# B&R Automation Studio project Panasonic_LinkaPowerCP2_A2021055 (part 16)

#### Main.st - Init, cyclic, exit code
```iecst
PROGRAM _INIT
	(* Insert code here *)

END_PROGRAM

PROGRAM _CYCLIC

	//Volanie funkcie SequenceControl//
	SequenceControl(SC:= SC_P2_StoperZaklTesnenia);

	//Volanie podprogramov//
	IOLinkKomunikacia;

	//Zhasnutie Bannera//
	IF P2_StoperZaklTesnenia.CMD.Banner_LED_OFF THEN
		P2_StoperZaklTesnenia.Banner.IN.ModraLED_ON:= FALSE;
		P2_StoperZaklTesnenia.Banner.IN.CervenaLED_ON:= FALSE;
		P2_StoperZaklTesnenia.Banner.IN.CyanLED_ON:= FALSE;
		P2_StoperZaklTesnenia.Banner.IN.ModraRotujucaLED_ON:= FALSE;
		P2_StoperZaklTesnenia.Banner.IN.OranzovaLED_ON:= FALSE;
		P2_StoperZaklTesnenia.Banner.IN.ZelenaLED_ON:= FALSE;
		P2_StoperZaklTesnenia.Banner.IN.ZltaLED_ON:= FALSE;
		P2_StoperZaklTesnenia.CMD.Banner_LED_OFF:= FALSE;
	END_IF

	//Reset sekcie //
	IF P2_StoperZaklTesnenia.Reset THEN
		SC_P2_StoperZaklTesnenia.Step:= 0;
		P2_StoperZaklTesnenia.Reset:= FALSE;
	ELSIF NOT Safety.STAV.Linka_ZonaCS_AKTIVNA THEN
		SC_P2_StoperZaklTesnenia.Step:= 0;
	END_IF

	CASE SC_P2_StoperZaklTesnenia.Step OF

		0:
			SC_P2_StoperZaklTesnenia.StepName:='0 - Nulovanie';
			P2_StoperZaklTesnenia.Automat:= FALSE;
			P2_StoperZaklTesnenia.KoniecCyklu:= FALSE;
			P2_StoperZaklTesnenia.Manual:= FALSE;
			P2_StoperZaklTesnenia.STAV.PoINIT:= FALSE;
			P2_StoperZaklTesnenia.OUT.ZasunStoper:= FALSE;
			P2_StoperZaklTesnenia.RFID_hlava.PrecitajChipRFID:= FALSE;
			P2_StoperZaklTesnenia.CMD.Banner_LED_OFF:= TRUE;
			P2_ZakladacTesnenia.COM_IN.ZalozTesnenie:= FALSE;
			P2_ZakladacTesnenia.COM_OUT.Stav_ZalozenieTesneniaUkoncene:= FALSE;
			CAM1.CMD.Triger:= FALSE;
			CAM1.STAV.Results_READY:= FALSE;
			FTP_CAM1.CMD.OdosliFotku:= FALSE;
			FTP_CAM1.CMD.VymazFotku:= FALSE;
			CAM7.CMD.Triger:= FALSE;
			CAM7.STAV.Results_READY:= FALSE;

			CAM8.CMD.Triger:= FALSE;
			CAM8.STAV.Results_READY:= FALSE;

			CAM17.CMD.Triger:= FALSE;
			CAM17.STAV.Results_READY:= FALSE;
			FTP_CAM17.CMD.OdosliFotku:= FALSE;
			FTP_CAM17.CMD.VymazFotku:= FALSE;
			P2_ZaklTesn_KAM_Result_Ignoruj:= FALSE;
			TRCB_P2_ZakladacTesnenia_ST3.CMD.VyziadajStavPaletky_TYP1:= FALSE;
			TRCB_P2_ZakladacTesnenia_ST3.CMD.PriradQRkodFiltra_TYP3:= FALSE;
			TRCB_P2_ZakladacTesnenia_ST3.CMD.OdosliStavPaletky_TYP2:= FALSE;
			TRCB_P2_ZakladacTesnenia_ST3.CMD.VyziadajStavPanatrace_TYP4:= FALSE;
			P2_Vizu.ZobrazHL1_ST3:= FALSE;
			P2_Vizu.ZobrazHL2_ST3:= FALSE;
			P2_Vizu.ZobrazHL3_ST3:= FALSE;
			P2_Vizu.ZobrazHL4_ST3:= FALSE;
			P2_Vizu.ZobrazHL5_ST3:= FALSE;
			P2_Vizu.ZobrazHL6_ST3:= FALSE;
			P2_Vizu.ZobrazHL7_ST3:= FALSE;
			P2_Vizu.ZobrazHL8_ST3:= FALSE;
			P2_Vizu.ZobrazHL9_ST3:= FALSE;
			P2_Vizu.ZobrazHL10_ST3:= FALSE;
			P2_Vizu.ZobrazHL11_ST3:= FALSE;
			P2_Vizu.ZobrazHL12_ST3:= FALSE;
			P2_Vizu.ZobrazHL14_ST3:= FALSE;
			P2_Vizu.ZobrazHL15_ST3:= FALSE;
			PocetDopytovNaServer:= 0;
			CisloFotky:= 0;
			PocetTrigrovKamery:= 0;
			P1_AkumulacnyStoper.STAV.PrebiehaVyvezeniePaletky:= FALSE;
			P2_StoperZaklTesnenia.STAV.PrebiehaVyvezeniePaletky:= FALSE;
			OpatovnaKontrolaFiltra_5H:= FALSE;
			PrecitanyQRkodPowerCP:= '';
			PrecitanyQRkodFiltra5H:= '';
			PrecitaneCisloPaletky:= '';
			TestovaciKus:= FALSE;
			P2_StoperZaklTesnenia.STAV.ObsluhaOznacilaPaletku_NG:= FALSE;
			P2_ZakladanieTesnenia_Taktime.IN.START_MeraniaCasu:= FALSE;
			P2_ZakladanieTesnenia_Taktime.IN.START_MeraniaStratovehoCasu:= FALSE;

			IF Safety.STAV.Linka_ZonaCS_AKTIVNA AND
				P2_Pracovisko.STAV.HardwareZaklTesnenia_OK AND
				NOT P2_Pracovisko.STAV.Porucha_ST1 THEN
				SC_P2_StoperZaklTesnenia.ResetStep:= TRUE;
				SC_P2_StoperZaklTesnenia.Step:= 1;
			END_IF

		1:
			SC_P2_StoperZaklTesnenia.StepName:='1 - Cakam na spustenie vyroby';
			P2_StoperZaklTesnenia.KoniecCyklu:= FALSE;
			IF P2_StoperZaklTesnenia.Automat THEN
				SC_P2_StoperZaklTesnenia.Step:= 2;
			ELSIF P2_StoperZaklTesnenia.Manual THEN
				SC_P2_StoperZaklTesnenia.Step:= 700;
			END_IF

			//********************************************************Inicializácia****************************************************************************//

		2:
			SC_P2_StoperZaklTesnenia.StepName:='2 - Inicializacia - cakam na spustenie inicializacie';
			SC_P2_StoperZaklTesnenia.IdleTime.PT:= T#4s;
			SC_P2_StoperZaklTesnenia.AlarmTime.PT:= T#5s;

			IF P2_ZakladacTesnenia.STAV.PoINIT AND P2_ZakladacTesnenia.ServoPojazduZakladaca.Status.ActPosition < 5  AND (*Safety.STAV.P2_ZaklTesn_PojazdMuting_AKTIVNY AND*) P2_Dopravniky.STAV.PoINIT THEN
				SC_P2_StoperZaklTesnenia.ResetStep:= TRUE;
				SC_P2_StoperZaklTesnenia.Step:= 3;
			END_IF

		3:
			SC_P2_StoperZaklTesnenia.StepName:='3 - Inicializacia - vymazanie adresarov kamier CAM1 a CAM 17';
			SC_P2_StoperZaklTesnenia.IdleTime.PT:= T#4s;
			SC_P2_StoperZaklTesnenia.AlarmTime.PT:= T#5s;

			P2_StoperZaklTesnenia.Banner.IN.ModraRotujucaLED_ON:= TRUE;

			IF NOT SC_P2_StoperZaklTesnenia.Switch1 THEN
				FTP_CAM1.CMD.VymazFotku:= TRUE;
				FTP_CAM17.CMD.VymazFotku:= TRUE;
				SC_P2_StoperZaklTesnenia.Switch1:= TRUE;
			END_IF

			IF FTP_CAM1.STATUS.KomunikaciaUkoncena AND FTP_CAM17.STATUS.KomunikaciaUkoncena THEN
				P2_StoperZaklTesnenia.CMD.Banner_LED_OFF:= TRUE;
				FTP_CAM1.CMD.VymazFotku:= FALSE;
				FTP_CAM17.CMD.VymazFotku:= FALSE;
				SC_P2_StoperZaklTesnenia.ResetStep:= TRUE;
				SC_P2_StoperZaklTesnenia.Step:= 5;
			ELSIF FTP_CAM1.STATUS.KomunikaciaError THEN
				P2_Alarmy[225]:= TRUE;
				P2_Pracovisko.STAV.Porucha_ST1:= TRUE;
			ELSIF FTP_CAM17.STATUS.KomunikaciaError THEN
				P2_Alarmy[228]:= TRUE;
				P2_Pracovisko.STAV.Porucha_ST1:= TRUE;
			END_IF

		5:
			SC_P2_StoperZaklTesnenia.StepName:='5 - Inicializacia - hladanie paletky na stopri';
			SC_P2_StoperZaklTesnenia.IdleTime.PT:= T#5s;
			SC_P2_StoperZaklTesnenia.AlarmTime.PT:= T#5s;

			SC_P2_StoperZaklTesnenia.IdleTime.IN:= TRUE;

			IF P2_StoperZaklTesnenia.RFID_hlava.PritomnostPaletky THEN
				SC_P2_StoperZaklTesnenia.ResetStep:= TRUE;
				SC_P2_StoperZaklTesnenia.Step:= 20;
			ELSIF SC_P2_StoperZaklTesnenia.IdleTime.Q THEN
				P2_StoperZaklTesnenia.STAV.PoINIT:= TRUE;
				SC_P2_StoperZaklTesnenia.ResetStep:= TRUE;
				SC_P2_StoperZaklTesnenia.Step:= 100;
			END_IF

		20:
			SC_P2_StoperZaklTesnenia.StepName:='20 - Inicializacia - precitanie cisla paletky';
			SC_P2_StoperZaklTesnenia.IdleTime.PT:= T#200ms;
			SC_P2_StoperZaklTesnenia.AlarmTime.PT:= T#5s;

			SC_P2_StoperZaklTesnenia.IdleTime.IN:= P2_StoperZaklTesnenia.RFID_hlava.PritomnostPaletky;

			IF SC_P2_StoperZaklTesnenia.IdleTime.Q AND NOT SC_P2_StoperZaklTesnenia.Switch1 THEN
				P2_StoperZaklTesnenia.RFID_hlava.PrecitajChipRFID:= TRUE;
				i:= 0;
				SC_P2_StoperZaklTesnenia.Switch1:= TRUE;
			END_IF

			IF P2_StoperZaklTesnenia.RFID_hlava.Stav_CitanieZapis_OK AND P2_StoperZaklTesnenia.RFID_hlava.PrecitaneCisloPaletky <> 0 THEN
				i:= P2_StoperZaklTesnenia.RFID_hlava.PrecitaneCisloPaletky;
				P2_StoperZaklTesnenia.PAR.CisloPaletky:= P2_StoperZaklTesnenia.RFID_hlava.PrecitaneCisloPaletky;
				P2_StoperZaklTesnenia.RFID_hlava.PrecitajChipRFID:= FALSE;
				SC_P2_StoperZaklTesnenia.ResetStep:= TRUE;
				SC_P2_StoperZaklTesnenia.Step:= 23;
			END_IF

		23:
			SC_P2_StoperZaklTesnenia.StepName:='23 - Inicializacia - kontrola a priradenie indexu paletky na zaklade precitanej hodnoty';
			SC_P2_StoperZaklTesnenia.IdleTime.PT:= T#200ms;
			SC_P2_StoperZaklTesnenia.AlarmTime.PT:= T#5s;

			IF i<> 0 THEN
				P2_StoperZaklTesnenia.PAR.CisloPaletky_STRING:= USINT_TO_STRING(i);
				Paletka[i].PAR.CisloPaletky:= USINT_TO_STRING(i);
				P2_ZakladacTesnenia.PAR.IndexPaletky:= i;
				SC_P2_StoperZaklTesnenia.ResetStep:= TRUE;
				SC_P2_StoperZaklTesnenia.Step:= 30;
			ELSE
				P2_Alarmy[200]:= TRUE;
				P2_Pracovisko.STAV.Porucha_ST1:= TRUE;
			END_IF

		30:
			SC_P2_StoperZaklTesnenia.StepName:='30 - Inicializacia - kontrola stavu paletky';
			SC_P2_StoperZaklTesnenia.IdleTime.PT:= T#200ms;
			SC_P2_StoperZaklTesnenia.AlarmTime.PT:= T#5s;

			IF Paletka[i].STAV.StavPaletky = '' THEN
				Paletka[i].STAV.StavPaletky:= 'NG';
				SC_P2_StoperZaklTesnenia.ResetStep:= TRUE;
				SC_P2_StoperZaklTesnenia.Step:= 560;
			ELSIF Paletka[i].STAV.StavPaletky = 'PRECH' THEN
				P2_StoperZaklTesnenia.STAV.PoINIT:= TRUE;
				SC_P2_StoperZaklTesnenia.ResetStep:= TRUE;
				SC_P2_StoperZaklTesnenia.Step:= 560;
			ELSIF Paletka[i].STAV.StavPaletky = 'TEST' AND Paletka[i].STAV.CisloTestovacejStanice = 'ST_3' THEN
				TestovaciKus:= TRUE;
			ELSIF Paletka[i].STAV.StavPaletky = 'TEST' AND Paletka[i].STAV.CisloTestovacejStanice <> 'ST_3' THEN
				P2_StoperZaklTesnenia.STAV.PoINIT:= TRUE;
				SC_P2_StoperZaklTesnenia.ResetStep:= TRUE;
				SC_P2_StoperZaklTesnenia.Step:= 560;
			ELSIF Paletka[i].STAV.StavPaletky = 'REV' AND Paletka[i].STAV.CisloRevorkovejStanice = 'ST_3' THEN
				Paletka[i].STAV.StavPaletky:= 'OK';
				SC_P2_StoperZaklTesnenia.ResetStep:= TRUE;
				SC_P2_StoperZaklTesnenia.Step:= 33;
			ELSIF Paletka[i].STAV.StavPaletky = 'REV' AND Paletka[i].STAV.CisloRevorkovejStanice <> 'ST_3' THEN
				P2_StoperZaklTesnenia.STAV.PoINIT:= TRUE;
				SC_P2_StoperZaklTesnenia.ResetStep:= TRUE;
				SC_P2_StoperZaklTesnenia.Step:= 560;
			ELSIF Paletka[i].STAV.StavPaletky = 'OK' THEN
				SC_P2_StoperZaklTesnenia.ResetStep:= TRUE;
				SC_P2_StoperZaklTesnenia.Step:= 33;
			ELSIF Paletka[i].STAV.StavPaletky = 'NG' THEN
				P2_StoperZaklTesnenia.STAV.PoINIT:= TRUE;
				SC_P2_StoperZaklTesnenia.ResetStep:= TRUE;
				SC_P2_StoperZaklTesnenia.Step:= 560;
			END_IF

		33:
			SC_P2_StoperZaklTesnenia.StepName:='33 - Inicializacia - kontrola uzavretia komunikacie';
			SC_P2_StoperZaklTesnenia.IdleTime.PT:= T#200ms;
			SC_P2_StoperZaklTesnenia.AlarmTime.PT:= T#5s;

			IF Paletka[i].STAV.Komunikacia_DONE THEN
				P2_StoperZaklTesnenia.STAV.PoINIT:= TRUE;
				SC_P2_StoperZaklTesnenia.ResetStep:= TRUE;
				SC_P2_StoperZaklTesnenia.Step:= 560;
			ELSE
				P2_StoperZaklTesnenia.STAV.PoINIT:= TRUE;
				SC_P2_StoperZaklTesnenia.ResetStep:= TRUE;
				SC_P2_StoperZaklTesnenia.Step:= 100;
			END_IF

			//********************************************************Automatický režim****************************************************************************//

		100:
			SC_P2_StoperZaklTesnenia.StepName:='100 - Automaticky Rezim - cakam na príchod paletky na stoper';
			SC_P2_StoperZaklTesnenia.IdleTime.PT:= T#200ms;
			SC_P2_StoperZaklTesnenia.AlarmTime.PT:= T#5s;

			SC_P2_StoperZaklTesnenia.IdleTime.IN:= P2_StoperZaklTesnenia.RFID_hlava.PritomnostPaletky;

			IF P2_StoperZaklTesnenia.RFID_hlava.PritomnostPaletky THEN
				P1_AkumulacnyStoper.STAV.PrebiehaVyvezeniePaletky:= FALSE;
			END_IF

			IF NOT SC_P2_StoperZaklTesnenia.Switch1 AND P2_StoperZaklTesnenia.RFID_hlava.PritomnostPaletky THEN
				P2_ZakladanieTesnenia_Taktime.IN.START_MeraniaCasu:= TRUE;
				P2_ZakladanieTesnenia_Taktime.IN.ZAPIS_MeraniaCasu:= TRUE;
				P2_ZakladanieTesnenia_Taktime.IN.ZAPIS_StratovyCas:= TRUE;
				Buffer_3.Hodnota:= P2_ZakladanieTesnenia_Taktime.OUT.StratoveSekundy;
				Buffer_3.ZapisHodnotu:= TRUE;
				SC_P2_StoperZaklTesnenia.Switch1:= TRUE;
			END_IF

			IF P2_StoperZaklTesnenia.KoniecCyklu THEN
				SC_P2_StoperZaklTesnenia.ResetStep:= TRUE;
				SC_P2_StoperZaklTesnenia.Step:= 0;
			ELSIF SC_P2_StoperZaklTesnenia.IdleTime.Q THEN
				SC_P2_StoperZaklTesnenia.ResetStep:= TRUE;
				SC_P2_StoperZaklTesnenia.Step:= 101;
			END_IF

		101:
			SC_P2_StoperZaklTesnenia.StepName:='101 - Automaticky Rezim - precitanie cisla paletky';
			SC_P2_StoperZaklTesnenia.IdleTime.PT:= T#500ms;
			SC_P2_StoperZaklTesnenia.AlarmTime.PT:= T#5s;
			SC_P2_StoperZaklTesnenia.IdleTime.IN:= TRUE;

			IF NOT SC_P2_StoperZaklTesnenia.Switch1 THEN
				i:= 0;
				P2_StoperZaklTesnenia.RFID_hlava.PrecitajChipRFID:= TRUE;
				SC_P2_StoperZaklTesnenia.Switch1:= TRUE;
			END_IF

			IF P2_StoperZaklTesnenia.RFID_hlava.Stav_CitanieZapis_OK AND P2_StoperZaklTesnenia.RFID_hlava.PrecitaneCisloPaletky <> 0 THEN
				i:= P2_StoperZaklTesnenia.RFID_hlava.PrecitaneCisloPaletky;
				P2_StoperZaklTesnenia.PAR.CisloPaletky:= P2_StoperZaklTesnenia.RFID_hlava.PrecitaneCisloPaletky;
				P2_StoperZaklTesnenia.RFID_hlava.PrecitajChipRFID:= FALSE;
				SC_P2_StoperZaklTesnenia.ResetStep:= TRUE;
				SC_P2_StoperZaklTesnenia.Step:= 102;
			END_IF

		102:
			SC_P2_StoperZaklTesnenia.StepName:='102 - Automaticky Rezim - kontrola a priradenie indexu paletky na zaklade precitanej hodnoty';
			SC_P2_StoperZaklTesnenia.IdleTime.PT:= T#200ms;
			SC_P2_StoperZaklTesnenia.AlarmTime.PT:= T#5s;

			IF i<> 0 THEN
				P2_StoperZaklTesnenia.PAR.CisloPaletky_STRING:= USINT_TO_STRING(i);
				Paletka[i].PAR.CisloPaletky:= USINT_TO_STRING(i);
				P2_ZakladacTesnenia.PAR.IndexPaletky:= i;
				SC_P2_StoperZaklTesnenia.ResetStep:= TRUE;
				SC_P2_StoperZaklTesnenia.Step:= 103;
			ELSE
				P2_Alarmy[200]:= TRUE;
				P2_Pracovisko.STAV.Porucha_ST1:= TRUE;
			END_IF

		103:
			SC_P2_StoperZaklTesnenia.StepName:='103 - Automaticky Rezim - kontrola stavu paletky';
			SC_P2_StoperZaklTesnenia.IdleTime.PT:= T#200ms;
			SC_P2_StoperZaklTesnenia.AlarmTime.PT:= T#5s;

			IF Paletka[i].STAV.StavPaletky = '' THEN
				Paletka[i].STAV.StavPaletky:= 'NG';
				SC_P2_StoperZaklTesnenia.ResetStep:= TRUE;
				SC_P2_StoperZaklTesnenia.Step:= 560;
			ELSIF Paletka[i].STAV.StavPaletky = 'PRECH' THEN
				SC_P2_StoperZaklTesnenia.ResetStep:= TRUE;
				SC_P2_StoperZaklTesnenia.Step:= 560;
			ELSIF Paletka[i].STAV.StavPaletky = 'TEST' AND Paletka[i].STAV.CisloTestovacejStanice = 'ST_3' THEN
				TestovaciKus:= TRUE;
			ELSIF Paletka[i].STAV.StavPaletky = 'TEST' AND Paletka[i].STAV.CisloTestovacejStanice <> 'ST_3' THEN
				SC_P2_StoperZaklTesnenia.ResetStep:= TRUE;
				SC_P2_StoperZaklTesnenia.Step:= 560;
			ELSIF Paletka[i].STAV.StavPaletky = 'REV' AND Paletka[i].STAV.CisloRevorkovejStanice = 'ST_3' THEN
				Paletka[i].STAV.StavPaletky:= 'OK';
				SC_P2_StoperZaklTesnenia.ResetStep:= TRUE;
				SC_P2_StoperZaklTesnenia.Step:= 105;
			ELSIF Paletka[i].STAV.StavPaletky = 'REV' AND Paletka[i].STAV.CisloRevorkovejStanice <> 'ST_3' THEN
				SC_P2_StoperZaklTesnenia.ResetStep:= TRUE;
				SC_P2_StoperZaklTesnenia.Step:= 560;
			ELSIF Paletka[i].STAV.StavPaletky = 'OK' THEN
				SC_P2_StoperZaklTesnenia.ResetStep:= TRUE;
				SC_P2_StoperZaklTesnenia.Step:= 105;
			ELSIF Paletka[i].STAV.StavPaletky = 'NG' THEN
				SC_P2_StoperZaklTesnenia.ResetStep:= TRUE;
				SC_P2_StoperZaklTesnenia.Step:= 560;
			END_IF

		105:
			SC_P2_StoperZaklTesnenia.StepName:='105 - Automaticky Rezim - vyziadanie stavu komunikacie zo serverom';
			SC_P2_StoperZaklTesnenia.IdleTime.PT:= T#200ms;
			SC_P2_StoperZaklTesnenia.AlarmTime.PT:= T#10s;

			P2_StoperZaklTesnenia.Banner.IN.ModraRotujucaLED_ON:= TRUE;

			IF Linka.KOM_Panatrace_OFF THEN
				P2_StoperZaklTesnenia.CMD.Banner_LED_OFF:= TRUE;
				SC_P2_StoperZaklTesnenia.ResetStep:= TRUE;
				SC_P2_StoperZaklTesnenia.Step:= 120;
			ELSIF NOT SC_P2_StoperZaklTesnenia.Switch1 AND TRCB_P2_ZakladacTesnenia_ST3.STATUS.KOM_READY THEN
				TRCB_P2_ZakladacTesnenia_ST3.CMD.VyziadajStavPanatrace_TYP4:= TRUE;
				(*P2_ZakladanieTesnenia_Taktime.IN.START_MeraniaStratovehoCasu:= TRUE;*)
				SC_P2_StoperZaklTesnenia.Switch1:= TRUE;
			END_IF

			IF TRCB_P2_ZakladacTesnenia_ST3.STATUS.KomunikaciaUkoncena THEN
				TRCB_P2_ZakladacTesnenia_ST3.CMD.VyziadajStavPanatrace_TYP4:= FALSE;
				P2_ZakladanieTesnenia_Taktime.IN.START_MeraniaStratovehoCasu:= FALSE;
				SC_P2_StoperZaklTesnenia.ResetStep:= TRUE;
				SC_P2_StoperZaklTesnenia.Step:= 106;
			ELSIF TRCB_P2_ZakladacTesnenia_ST3.STATUS.KomunikaciaError THEN
				P2_StoperZaklTesnenia.CMD.Banner_LED_OFF:= TRUE;
				TRCB_P2_ZakladacTesnenia_ST3.CMD.VyziadajStavPanatrace_TYP4:= FALSE;
				P2_ZakladanieTesnenia_Taktime.IN.START_MeraniaStratovehoCasu:= FALSE;
				SC_P2_StoperZaklTesnenia.ResetStep:= TRUE;
				SC_P2_StoperZaklTesnenia.Step:= 107;
			END_IF

		106:
			SC_P2_StoperZaklTesnenia.StepName:='106 - Automaticky Rezim - kontrola odpovede servera';
			SC_P2_StoperZaklTesnenia.IdleTime.PT:= T#200ms;
			SC_P2_StoperZaklTesnenia.AlarmTime.PT:= T#5s;

			IF NOT TRCB_P2_ZakladacTesnenia_ST3.STATUS.KomunikaciaUkoncena THEN
				IF TRCB_P2_ZakladacTesnenia_ST3.OUTPUTS.DruhCinnostiNaPaletke = '0;Generating' THEN
					SC_P2_StoperZaklTesnenia.ResetStep:= TRUE;
					SC_P2_StoperZaklTesnenia.Step:= 107;
				ELSIF TRCB_P2_ZakladacTesnenia_ST3.OUTPUTS.DruhCinnostiNaPaletke = '1;Request' THEN
					SC_P2_StoperZaklTesnenia.ResetStep:= TRUE;
					SC_P2_StoperZaklTesnenia.Step:= 108;
				ELSIF TRCB_P2_ZakladacTesnenia_ST3.OUTPUTS.DruhCinnostiNaPaletke = '2;Report' THEN
					SC_P2_StoperZaklTesnenia.ResetStep:= TRUE;
					SC_P2_StoperZaklTesnenia.Step:= 160;
				ELSIF TRCB_P2_ZakladacTesnenia_ST3.OUTPUTS.DruhCinnostiNaPaletke = '3;Wedding' THEN
					SC_P2_StoperZaklTesnenia.ResetStep:= TRUE;
					SC_P2_StoperZaklTesnenia.Step:= 130;
				ELSIF TRCB_P2_ZakladacTesnenia_ST3.OUTPUTS.DruhCinnostiNaPaletke = '4;Status' THEN
					SC_P2_StoperZaklTesnenia.ResetStep:= TRUE;
					SC_P2_StoperZaklTesnenia.Step:= 107;
				ELSIF TRCB_P2_ZakladacTesnenia_ST3.OUTPUTS.DruhCinnostiNaPaletke = '5;' THEN
					SC_P2_StoperZaklTesnenia.ResetStep:= TRUE;
					SC_P2_StoperZaklTesnenia.Step:= 107;
				ELSE
					SC_P2_StoperZaklTesnenia.ResetStep:= TRUE;
					SC_P2_StoperZaklTesnenia.Step:= 107;
				END_IF
			END_IF

		107:
			SC_P2_StoperZaklTesnenia.StepName:='107 - Automaticky Rezim - rozhodnutie obsluhy po chybe komunikacie s Panatrace';
			SC_P2_StoperZaklTesnenia.IdleTime.PT:= T#200ms;
			SC_P2_StoperZaklTesnenia.AlarmTime.PT:= T#5s;

			P2_StoperZaklTesnenia.CMD.Banner_LED_OFF:= TRUE;
			P2_Vizu.ZobrazHL15_ST3:= TRUE;

			IF TRCB_P2_ZaklTesn_OpatovnyDopyt THEN
				TRCB_P2_ZaklTesn_OpatovnyDopyt:= FALSE;
				P2_Vizu.ZobrazHL15_ST3:= FALSE;
				SC_P2_StoperZaklTesnenia.ResetStep:= TRUE;
				SC_P2_StoperZaklTesnenia.Step:= 105;
			ELSIF TRCB_P2_ZaklTesn_PaletkaNG THEN
				TRCB_P2_ZaklTesn_PaletkaNG:= FALSE;
				P2_Vizu.ZobrazHL15_ST3:= FALSE;
				Paletka[i].STAV.StavPaletky := 'NG';
				SC_P2_StoperZaklTesnenia.ResetStep:= TRUE;
				SC_P2_StoperZaklTesnenia.Step:= 560;
			END_IF

		108:
			SC_P2_StoperZaklTesnenia.StepName:='108 - Automaticky Rezim - vyziadanie stavu paletky zo servera';
			SC_P2_StoperZaklTesnenia.IdleTime.PT:= T#200ms;
			SC_P2_StoperZaklTesnenia.AlarmTime.PT:= T#10s;
			SC_P2_StoperZaklTesnenia.IdleTime.IN:= TRUE;

			IF NOT SC_P2_StoperZaklTesnenia.Switch1 AND TRCB_P2_ZakladacTesnenia_ST3.STATUS.KOM_READY THEN
				TRCB_P2_ZakladacTesnenia_ST3.CMD.VyziadajStavPaletky_TYP1:= TRUE;
				(*P2_ZakladanieTesnenia_Taktime.IN.START_MeraniaStratovehoCasu:= TRUE;*)
				SC_P2_StoperZaklTesnenia.Switch1:= TRUE;
			END_IF

			IF TRCB_P2_ZakladacTesnenia_ST3.STATUS.KomunikaciaUkoncena THEN
				P2_StoperZaklTesnenia.CMD.Banner_LED_OFF:= TRUE;
				TRCB_P2_ZakladacTesnenia_ST3.CMD.VyziadajStavPaletky_TYP1:= FALSE;
				P2_ZakladanieTesnenia_Taktime.IN.START_MeraniaStratovehoCasu:= FALSE;
				SC_P2_StoperZaklTesnenia.ResetStep:= TRUE;
				SC_P2_StoperZaklTesnenia.Step:= 110;
			ELSIF TRCB_P2_ZakladacTesnenia_ST3.STATUS.KomunikaciaError THEN
				P2_StoperZaklTesnenia.CMD.Banner_LED_OFF:= TRUE;
				TRCB_P2_ZakladacTesnenia_ST3.CMD.VyziadajStavPaletky_TYP1:= FALSE;
				P2_ZakladanieTesnenia_Taktime.IN.START_MeraniaStratovehoCasu:= FALSE;
				SC_P2_StoperZaklTesnenia.ResetStep:= TRUE;
				SC_P2_StoperZaklTesnenia.Step:= 115;
			END_IF

		110:
			SC_P2_StoperZaklTesnenia.StepName:='110 - Automaticky Rezim - kontrola odpovede servera';
			SC_P2_StoperZaklTesnenia.IdleTime.PT:= T#200ms;
			SC_P2_StoperZaklTesnenia.AlarmTime.PT:= T#5s;

			IF NOT TRCB_P2_ZakladacTesnenia_ST3.STATUS.KomunikaciaUkoncena THEN
				IF TRCB_P2_ZakladacTesnenia_ST3.OUTPUTS.PovolenieCinnostiNaPaletke = 'OK' THEN
					IF TRCB_P2_ZakladacTesnenia_ST3.OUTPUTS.DruhCinnostiNaPaletke = 'PRD;ST3' THEN
						IF NOT OpatovnaKontrolaFiltra_5H THEN
							SC_P2_StoperZaklTesnenia.ResetStep:= TRUE;
							SC_P2_StoperZaklTesnenia.Step:= 120;
						ELSE
							CAM7.STAV.Results_READY:= FALSE;
							SC_P2_StoperZaklTesnenia.ResetStep:= TRUE;
							SC_P2_StoperZaklTesnenia.Step:= 130;
						END_IF
					END_IF
				ELSIF TRCB_P2_ZakladacTesnenia_ST3.OUTPUTS.PovolenieCinnostiNaPaletke = 'NG' THEN
					SC_P2_StoperZaklTesnenia.ResetStep:= TRUE;
					SC_P2_StoperZaklTesnenia.Step:= 115;
				END_IF
			END_IF

		115:
			SC_P2_StoperZaklTesnenia.StepName:='115 - Automaticky Rezim - rozhodnutie obsluhy po odpovedi panatrace NG';
			SC_P2_StoperZaklTesnenia.IdleTime.PT:= T#200ms;
			SC_P2_StoperZaklTesnenia.AlarmTime.PT:= T#5s;

			P2_Vizu.ZobrazHL13_ST3:= TRUE;

			IF TRCB_P2_ZaklTesn_OpatovnyDopyt THEN
				TRCB_P2_ZaklTesn_OpatovnyDopyt:= FALSE;
				P2_Vizu.ZobrazHL13_ST3:= FALSE;
				SC_P2_StoperZaklTesnenia.ResetStep:= TRUE;
				SC_P2_StoperZaklTesnenia.Step:= 105;
			ELSIF TRCB_P2_ZaklTesn_PaletkaNG THEN
				TRCB_P2_ZaklTesn_PaletkaNG:= FALSE;
				P2_Vizu.ZobrazHL13_ST3:= FALSE;
				Paletka[i].STAV.StavPaletky := 'NG';
				SC_P2_StoperZaklTesnenia.ResetStep:= TRUE;
				SC_P2_StoperZaklTesnenia.Step:= 560;
			END_IF

		120:
			SC_P2_StoperZaklTesnenia.StepName:='120 - Automaticky Rezim - vystavenie signalu pre zakladac,zaloz tesnenie';
			SC_P2_StoperZaklTesnenia.IdleTime.PT:= T#200ms;
			SC_P2_StoperZaklTesnenia.AlarmTime.PT:= T#5s;

			IF NOT SC_P2_StoperZaklTesnenia.Switch1 THEN
				P2_ZakladacTesnenia.COM_IN.ZalozTesnenie:= TRUE;
				SC_P2_StoperZaklTesnenia.Switch1:= TRUE;
			END_IF

			IF P2_ZakladacTesnenia.COM_OUT.Stav_ZalozenieTesneniaUkoncene THEN
				P2_StoperZaklTesnenia.Banner.IN.ZelenaLED_ON:= TRUE;
			END_IF

			IF P2_StoperZaklTesnenia.KoniecCyklu AND NOT P2_ZakladacTesnenia.Automat THEN
				SC_P2_StoperZaklTesnenia.ResetStep:= TRUE;
				SC_P2_StoperZaklTesnenia.Step:= 0;
			ELSIF P2_ZakladacTesnenia.COM_OUT.Stav_ZalozenieTesneniaUkoncene AND NOT P2_ZakladacTesnenia.IN.Pojazd_PritomPowerCP AND NOT P2_StoperZaklTesnenia.STAV.ObsluhaOznacilaPaletku_NG THEN
				P2_ZakladacTesnenia.COM_OUT.Stav_ZalozenieTesneniaUkoncene:= FALSE;
				P2_ZakladacTesnenia.COM_IN.ZalozTesnenie:= FALSE;
				P2_StoperZaklTesnenia.CMD.Banner_LED_OFF:= TRUE;
				SC_P2_StoperZaklTesnenia.ResetStep:= TRUE;
				SC_P2_StoperZaklTesnenia.Step:= 130;
			ELSIF P2_ZakladacTesnenia.COM_OUT.Stav_ZalozenieTesneniaUkoncene AND NOT P2_ZakladacTesnenia.IN.Pojazd_PritomPowerCP AND P2_StoperZaklTesnenia.STAV.ObsluhaOznacilaPaletku_NG THEN
				P2_ZakladacTesnenia.COM_IN.ZalozTesnenie:= FALSE;
				P2_StoperZaklTesnenia.CMD.Banner_LED_OFF:= TRUE;
				SC_P2_StoperZaklTesnenia.ResetStep:= TRUE;
				SC_P2_StoperZaklTesnenia.Step:= 125;
			END_IF

		125:
			SC_P2_StoperZaklTesnenia.StepName:='125 - Automaticky Rezim - rozhodnutie po oznaceni paletky ako NG';
			SC_P2_StoperZaklTesnenia.IdleTime.PT:= T#200ms;
			SC_P2_StoperZaklTesnenia.AlarmTime.PT:= T#5s;

			IF Linka.PAR.ZvolenyModel = '5H' THEN
				Paletka[i].PAR.StavPowerCP:= 'FAIL';
				Paletka[i].STAV.StavPaletky := 'NG';
				SC_P2_StoperZaklTesnenia.ResetStep:= TRUE;
				SC_P2_StoperZaklTesnenia.Step:= 140;
			ELSE
				Paletka[i].PAR.StavPowerCP:= 'FAIL';
				Paletka[i].STAV.StavPaletky := 'NG';
				SC_P2_StoperZaklTesnenia.ResetStep:= TRUE;
				SC_P2_StoperZaklTesnenia.Step:= 550;
			END_IF

		130:
			SC_P2_StoperZaklTesnenia.StepName:='130 - Automaticky Rezim - kontrola typu modelu';
			SC_P2_StoperZaklTesnenia.IdleTime.PT:= T#200ms;
			SC_P2_StoperZaklTesnenia.AlarmTime.PT:= T#5s;

			IF Linka.PAR.ZvolenyModel = '5H' THEN
				CAM7.STAV.OldRunCounter:= CAM7.STAV.RunCounter;
				CAM7.STAV.Results_READY:= FALSE;
				SC_P2_StoperZaklTesnenia.ResetStep:= TRUE;
				SC_P2_StoperZaklTesnenia.Step:= 132;
			ELSE
				SC_P2_StoperZaklTesnenia.ResetStep:= TRUE;
				SC_P2_StoperZaklTesnenia.Step:= 160;
			END_IF

		132:
			SC_P2_StoperZaklTesnenia.StepName:='132 - Automaticky Rezim - kamerova kontrola pritomnosti filtra 5H v drziaku filtra CAM7';//CAM 7 - iba model 5H//
			SC_P2_StoperZaklTesnenia.IdleTime.PT:= T#5s;
			SC_P2_StoperZaklTesnenia.AlarmTime.PT:= T#5s;

			P2_StoperZaklTesnenia.Banner.IN.ModraLED_ON:= TRUE;

			IF NOT SC_P2_StoperZaklTesnenia.Switch1 AND CAM7.STAV.Command_READY THEN
				CAM7.CMD.Triger:= TRUE;
				SC_P2_StoperZaklTesnenia.IdleTime.IN:= TRUE;
				SC_P2_StoperZaklTesnenia.Switch1:= TRUE;
			END_IF

			IF CAM7.STAV.Results_READY AND CAM7.STAV.Command_AKCEPTOVANY AND CAM7.STAV.OldRunCounter <> CAM7.STAV.RunCounter  THEN
				PocetTrigrovKamery:= 0;
				CAM7.STAV.Results_READY:= FALSE;
				CAM7.STAV.OldRunCounter:= CAM7.STAV.RunCounter;
				P2_StoperZaklTesnenia.CMD.Banner_LED_OFF:= TRUE;
				SC_P2_StoperZaklTesnenia.ResetStep:= TRUE;
				SC_P2_StoperZaklTesnenia.Step:= 134;
			ELSIF SC_P2_StoperZaklTesnenia.IdleTime.Q AND PocetTrigrovKamery < 5 THEN
				PocetTrigrovKamery:= PocetTrigrovKamery + 1;
				CAM7.STAV.Results_READY:= FALSE;
				CAM7.STAV.OldRunCounter:= CAM7.STAV.RunCounter;
				CAM7.CMD.Triger:= FALSE;
				P2_StoperZaklTesnenia.CMD.Banner_LED_OFF:= TRUE;
				SC_P2_StoperZaklTesnenia.ResetStep:= TRUE;
				SC_P2_StoperZaklTesnenia.Step:= 133;
			ELSIF SC_P2_StoperZaklTesnenia.IdleTime.Q AND PocetTrigrovKamery >= 5 THEN
				P2_Alarmy[291]:= TRUE;
				P2_Pracovisko.STAV.Porucha_ST1:= TRUE;
			END_IF

		133:
			SC_P2_StoperZaklTesnenia.StepName:='133 - Automaticky Rezim - cakam na opatovny triger kamery CAM7';
			SC_P2_StoperZaklTesnenia.IdleTime.PT:= T#1s;
			SC_P2_StoperZaklTesnenia.AlarmTime.PT:= T#5s;
			SC_P2_StoperZaklTesnenia.IdleTime.IN:= TRUE;

			IF SC_P2_StoperZaklTesnenia.IdleTime.Q THEN
				SC_P2_StoperZaklTesnenia.ResetStep:= TRUE;
				SC_P2_StoperZaklTesnenia.Step:= 132;
			END_IF

		134:
			SC_P2_StoperZaklTesnenia.StepName:='134 - Automaticky Rezim - vysledok kamerovej kontroly filtra 5H';
			SC_P2_StoperZaklTesnenia.IdleTime.PT:= T#500ms;
			SC_P2_StoperZaklTesnenia.AlarmTime.PT:= T#5s;
			SC_P2_StoperZaklTesnenia.IdleTime.IN:= TRUE;

			IF Linka.P2_Kamery_OFF THEN
				CAM7.CMD.Triger:= FALSE;
				CAM7.PAR.ResultFotky:= 'PASS';
				SC_P2_StoperZaklTesnenia.ResetStep:= TRUE;
				SC_P2_StoperZaklTesnenia.Step:= 135;
			ELSIF NOT CAM7.STAV.BUSY THEN
				CAM7.CMD.Triger:= FALSE;
				IF P2_StoperZaklTesnenia.STAV.ObsluhaOznacilaPaletku_NG THEN
					CAM7.PAR.ResultFotky:= 'FAIL';
					SC_P2_StoperZaklTesnenia.ResetStep:= TRUE;
					SC_P2_StoperZaklTesnenia.Step:= 180;
				ELSIF CAM7.RESULT.CitanieQRkodu_Filtra5H_OK THEN
					IF P2_StoperZaklTesnenia.PAR.StaryQRkod_Filtra5H <> CAM7.RESULT.PrecitanyQRkod_Filtra5H THEN
						Paletka[i].PAR.QRkodFiltra_5H:= CAM7.RESULT.PrecitanyQRkod_Filtra5H;
						CAM7.PAR.ResultFotky:= 'PASS';
						SC_P2_StoperZaklTesnenia.ResetStep:= TRUE;
						SC_P2_StoperZaklTesnenia.Step:= 135;
					ELSE
						CAM7.PAR.ResultFotky:= 'FAIL';
						SC_P2_StoperZaklTesnenia.ResetStep:= TRUE;
						SC_P2_StoperZaklTesnenia.Step:= 135;
					END_IF
				ELSE
					CAM7.PAR.ResultFotky:= 'FAIL';
					SC_P2_StoperZaklTesnenia.ResetStep:= TRUE;
					SC_P2_StoperZaklTesnenia.Step:= 135;
				END_IF
			END_IF

		135:
			SC_P2_StoperZaklTesnenia.StepName:='135 - Automaticky Rezim - rozhodnutie podla kamerovej kontroly filtra 5H';
			SC_P2_StoperZaklTesnenia.IdleTime.PT:= T#200ms;
			SC_P2_StoperZaklTesnenia.AlarmTime.PT:= T#5s;

			IF CAM7.PAR.ResultFotky = 'PASS' THEN
				SC_P2_StoperZaklTesnenia.ResetStep:= TRUE;
				SC_P2_StoperZaklTesnenia.Step:= 140;
			ELSIF CAM7.PAR.ResultFotky = 'FAIL' THEN
				SC_P2_StoperZaklTesnenia.ResetStep:= TRUE;
				SC_P2_StoperZaklTesnenia.Step:= 137;
			END_IF

		137:
			SC_P2_StoperZaklTesnenia.StepName:='137 - Automaticky Rezim - zobrazenie hlasenia neprecitany QR kod filtra 5H';
			SC_P2_StoperZaklTesnenia.IdleTime.PT:= T#200ms;
			SC_P2_StoperZaklTesnenia.AlarmTime.PT:= T#5s;

			IF NOT SC_P2_StoperZaklTesnenia.Switch1 THEN
				P2_Vizu.ZobrazHL4_ST3:= TRUE;
				SC_P2_StoperZaklTesnenia.Switch1:= TRUE;
			END_IF

			P2_StoperZaklTesnenia.Banner.IN.CervenaLED_ON:= Blikac500ms;

			IF P2_StoperZaklTesnenia.Banner.OUT.Stlaceny THEN
				CAM7.STAV.Results_READY:= FALSE;
				P2_Vizu.ZobrazHL4_ST3:= FALSE;
				P2_StoperZaklTesnenia.CMD.Banner_LED_OFF:= TRUE;
				SC_P2_StoperZaklTesnenia.ResetStep:= TRUE;
				SC_P2_StoperZaklTesnenia.Step:= 132;
			END_IF

		140:
			SC_P2_StoperZaklTesnenia.StepName:='140 - Automaticky Rezim - vyziadanie stavu komunikacie zo serverom';
			SC_P2_StoperZaklTesnenia.IdleTime.PT:= T#200ms;
			SC_P2_StoperZaklTesnenia.AlarmTime.PT:= T#10s;

			P2_StoperZaklTesnenia.Banner.IN.ModraRotujucaLED_ON:= TRUE;

			IF Linka.KOM_Panatrace_OFF THEN
				P2_StoperZaklTesnenia.CMD.Banner_LED_OFF:= TRUE;
				SC_P2_StoperZaklTesnenia.ResetStep:= TRUE;
				SC_P2_StoperZaklTesnenia.Step:= 160;
			ELSE
				SC_P2_StoperZaklTesnenia.ResetStep:= TRUE;
				SC_P2_StoperZaklTesnenia.Step:= 145;
			END_IF
			//			ELSIF NOT SC_P2_StoperZaklTesnenia.Switch1 THEN
			//				TRCB_P2_ZakladacTesnenia_ST3.CMD.VyziadajStavPanatrace_TYP4:= TRUE;
			//				SC_P2_StoperZaklTesnenia.Switch1:= TRUE;
			//			END_IF
			//
			//			IF TRCB_P2_ZakladacTesnenia_ST3.STATUS.KomunikaciaUkoncena THEN
			//				P2_StoperZaklTesnenia.CMD.Banner_LED_OFF:= TRUE;
			//				TRCB_P2_ZakladacTesnenia_ST3.CMD.VyziadajStavPanatrace_TYP4:= FALSE;
			//				SC_P2_StoperZaklTesnenia.ResetStep:= TRUE;
			//				SC_P2_StoperZaklTesnenia.Step:= 141;
			//			ELSIF TRCB_P2_ZakladacTesnenia_ST3.STATUS.KomunikaciaError THEN
			//				P2_Alarmy[230]:= TRUE;
			//				P2_Pracovisko.STAV.Porucha_ST1:= TRUE;
			//			END_IF

		141:
			SC_P2_StoperZaklTesnenia.StepName:='141 - Automaticky Rezim - kontrola odpovede servera';
			SC_P2_StoperZaklTesnenia.IdleTime.PT:= T#200ms;
			SC_P2_StoperZaklTesnenia.AlarmTime.PT:= T#5s;

			IF NOT TRCB_P2_ZakladacTesnenia_ST3.STATUS.KomunikaciaUkoncena THEN
				IF TRCB_P2_ZakladacTesnenia_ST3.OUTPUTS.DruhCinnostiNaPaletke = '0;Generating' THEN
					SC_P2_StoperZaklTesnenia.ResetStep:= TRUE;
					SC_P2_StoperZaklTesnenia.Step:= 142;
				ELSIF TRCB_P2_ZakladacTesnenia_ST3.OUTPUTS.DruhCinnostiNaPaletke = '1;Request' THEN
					SC_P2_StoperZaklTesnenia.ResetStep:= TRUE;
					SC_P2_StoperZaklTesnenia.Step:= 142;
				ELSIF TRCB_P2_ZakladacTesnenia_ST3.OUTPUTS.DruhCinnostiNaPaletke = '2;Report' THEN
					SC_P2_StoperZaklTesnenia.ResetStep:= TRUE;
					SC_P2_StoperZaklTesnenia.Step:= 160;
				ELSIF TRCB_P2_ZakladacTesnenia_ST3.OUTPUTS.DruhCinnostiNaPaletke = '3;Wedding' THEN
					SC_P2_StoperZaklTesnenia.ResetStep:= TRUE;
					SC_P2_StoperZaklTesnenia.Step:= 145;
				ELSIF TRCB_P2_ZakladacTesnenia_ST3.OUTPUTS.DruhCinnostiNaPaletke = '4;Status' THEN
					SC_P2_StoperZaklTesnenia.ResetStep:= TRUE;
					SC_P2_StoperZaklTesnenia.Step:= 142;
				ELSIF TRCB_P2_ZakladacTesnenia_ST3.OUTPUTS.DruhCinnostiNaPaletke = '5;' THEN
					SC_P2_StoperZaklTesnenia.ResetStep:= TRUE;
					SC_P2_StoperZaklTesnenia.Step:= 142;
				END_IF
			END_IF

		142:
			SC_P2_StoperZaklTesnenia.StepName:='142 - Automaticky Rezim - rozhodnutie obsluhy po chybe komunikacie s Panatrace';
			SC_P2_StoperZaklTesnenia.IdleTime.PT:= T#200ms;
			SC_P2_StoperZaklTesnenia.AlarmTime.PT:= T#5s;

			P2_Vizu.ZobrazHL15_ST3:= TRUE;

			IF TRCB_P2_ZaklTesn_OpatovnyDopyt THEN
				TRCB_P2_ZaklTesn_OpatovnyDopyt:= FALSE;
				P2_Vizu.ZobrazHL15_ST3:= FALSE;
				SC_P2_StoperZaklTesnenia.ResetStep:= TRUE;
				SC_P2_StoperZaklTesnenia.Step:= 140;
			ELSIF TRCB_P2_ZaklTesn_PaletkaNG THEN
				TRCB_P2_ZaklTesn_PaletkaNG:= FALSE;
				P2_Vizu.ZobrazHL15_ST3:= FALSE;
				Paletka[i].STAV.StavPaletky := 'NG';
				SC_P2_StoperZaklTesnenia.ResetStep:= TRUE;
				SC_P2_StoperZaklTesnenia.Step:= 560;
			END_IF

		145:
			SC_P2_StoperZaklTesnenia.StepName:='145 - Automaticky Rezim - priradenie QRkodu filtra';
			SC_P2_StoperZaklTesnenia.IdleTime.PT:= T#200ms;
			SC_P2_StoperZaklTesnenia.AlarmTime.PT:= T#10s;
			SC_P2_StoperZaklTesnenia.IdleTime.IN:= TRUE;

			P2_StoperZaklTesnenia.Banner.IN.ModraRotujucaLED_ON:= TRUE;

			IF NOT SC_P2_StoperZaklTesnenia.Switch1 AND TRCB_P2_ZakladacTesnenia_ST3.STATUS.KOM_READY THEN
				TRCB_P2_ZakladacTesnenia_ST3.CMD.PriradQRkodFiltra_TYP3:= TRUE;
				(*P2_ZakladanieTesnenia_Taktime.IN.START_MeraniaStratovehoCasu:= TRUE;*)
				SC_P2_StoperZaklTesnenia.Switch1:= TRUE;
			END_IF

			IF TRCB_P2_ZakladacTesnenia_ST3.STATUS.KomunikaciaUkoncena THEN
				P2_StoperZaklTesnenia.CMD.Banner_LED_OFF:= TRUE;
				TRCB_P2_ZakladacTesnenia_ST3.CMD.PriradQRkodFiltra_TYP3:= FALSE;
				P2_ZakladanieTesnenia_Taktime.IN.START_MeraniaStratovehoCasu:= FALSE;
				SC_P2_StoperZaklTesnenia.ResetStep:= TRUE;
				SC_P2_StoperZaklTesnenia.Step:= 148;
			ELSIF TRCB_P2_ZakladacTesnenia_ST3.STATUS.KomunikaciaError THEN
				TRCB_P2_ZakladacTesnenia_ST3.CMD.PriradQRkodFiltra_TYP3:= FALSE;
				P2_ZakladanieTesnenia_Taktime.IN.START_MeraniaStratovehoCasu:= FALSE;
				P2_Alarmy[230]:= TRUE;
				P2_Pracovisko.STAV.Porucha_ST1:= TRUE;
			END_IF

		148:
			SC_P2_StoperZaklTesnenia.StepName:='148 - Automaticky Rezim - kontrola odpovede servera';
			SC_P2_StoperZaklTesnenia.IdleTime.PT:= T#200ms;
			SC_P2_StoperZaklTesnenia.AlarmTime.PT:= T#10s;

			IF NOT TRCB_P2_ZakladacTesnenia_ST3.STATUS.KomunikaciaUkoncena THEN
				IF P2_StoperZaklTesnenia.STAV.ObsluhaOznacilaPaletku_NG THEN
					SC_P2_StoperZaklTesnenia.ResetStep:= TRUE;
					SC_P2_StoperZaklTesnenia.Step:= 180;
				ELSIF TRCB_P2_ZakladacTesnenia_ST3.OUTPUTS.PovolenieCinnostiNaPaletke = 'OK' THEN
					Paletka[i].STAV.QRkodFiltraPriradeny:= TRUE;
					OpatovnaKontrolaFiltra_5H:= FALSE;
					Paletka[i].PAR.StavPowerCP:= 'PASS';
					SC_P2_StoperZaklTesnenia.ResetStep:= TRUE;
					SC_P2_StoperZaklTesnenia.Step:= 160;
				ELSIF TRCB_P2_ZakladacTesnenia_ST3.OUTPUTS.PovolenieCinnostiNaPaletke = 'NG' THEN
					Paletka[i].STAV.QRkodFiltraPriradeny:= FALSE;
					IF P2_StoperZaklTesnenia.STAV.ObsluhaOznacilaPaletku_NG THEN
						SC_P2_StoperZaklTesnenia.ResetStep:= TRUE;
						SC_P2_StoperZaklTesnenia.Step:= 560;
					ELSE
						SC_P2_StoperZaklTesnenia.ResetStep:= TRUE;
						SC_P2_StoperZaklTesnenia.Step:= 150;
					END_IF
				END_IF
			END_IF

		150:
			SC_P2_StoperZaklTesnenia.StepName:='150 - Automaticky Rezim - zobrazenie hlasenia nespravny typ Filtra';
			SC_P2_StoperZaklTesnenia.IdleTime.PT:= T#200ms;
			SC_P2_StoperZaklTesnenia.AlarmTime.PT:= T#10s;

			P2_StoperZaklTesnenia.Banner.IN.CervenaLED_ON:= Blikac500ms;

			IF NOT SC_P2_StoperZaklTesnenia.Switch1 THEN
				P2_Vizu.ZobrazHL9_ST3:= TRUE;
				SC_P2_StoperZaklTesnenia.Switch1:= TRUE;
			END_IF

			IF P2_StoperZaklTesnenia.Banner.OUT.Stlaceny THEN
				P2_Vizu.ZobrazHL9_ST3:= FALSE;
				P2_StoperZaklTesnenia.CMD.Banner_LED_OFF:= TRUE;
				SC_P2_StoperZaklTesnenia.ResetStep:= TRUE;
				SC_P2_StoperZaklTesnenia.Step:= 153;
			END_IF

		153:
			SC_P2_StoperZaklTesnenia.StepName:='153 - Automaticky Rezim - vymazanie adresarov kamier CAM1 ';
			SC_P2_StoperZaklTesnenia.IdleTime.PT:= T#4s;
			SC_P2_StoperZaklTesnenia.AlarmTime.PT:= T#5s;

			IF Linka.KOM_FTP_OFF THEN
				SC_P2_StoperZaklTesnenia.ResetStep:= TRUE;
				SC_P2_StoperZaklTesnenia.Step:= 105;
			ELSIF NOT SC_P2_StoperZaklTesnenia.Switch1 THEN
				FTP_CAM1.CMD.VymazFotku:= TRUE;
				SC_P2_StoperZaklTesnenia.Switch1:= TRUE;
			END_IF

			IF FTP_CAM1.STATUS.KomunikaciaUkoncena THEN
				OpatovnaKontrolaFiltra_5H:= TRUE;
				FTP_CAM1.CMD.VymazFotku:= FALSE;
				SC_P2_StoperZaklTesnenia.ResetStep:= TRUE;
				SC_P2_StoperZaklTesnenia.Step:= 105;
			ELSIF FTP_CAM1.STATUS.KomunikaciaError THEN
				P2_Alarmy[225]:= TRUE;
				P2_Pracovisko.STAV.Porucha_ST1:= TRUE;
			END_IF

		160:
			SC_P2_StoperZaklTesnenia.StepName:='160 - Automaticky Rezim - cakam na potvrdenie bannera, kontrola prihlasenia operatora';
			SC_P2_StoperZaklTesnenia.IdleTime.PT:= T#200ms;
			SC_P2_StoperZaklTesnenia.AlarmTime.PT:= T#5s;

			IF P2_UzivatelPrihlaseny THEN
				P2_Vizu.ZobrazHL12_ST3:= FALSE;
				P2_StoperZaklTesnenia.Banner.IN.ZelenaLED_ON:= TRUE;
				P2_StoperZaklTesnenia.Banner.IN.CyanLED_ON:= FALSE;
			ELSE
				P2_Vizu.ZobrazHL12_ST3:= TRUE;
				P2_StoperZaklTesnenia.Banner.IN.ZelenaLED_ON:= FALSE;
				P2_StoperZaklTesnenia.Banner.IN.CyanLED_ON:= Blikac500ms;
			END_IF

			IF P2_StoperZaklTesnenia.KoniecCyklu THEN
				SC_P2_StoperZaklTesnenia.ResetStep:= TRUE;
				SC_P2_StoperZaklTesnenia.Step:= 0;
			ELSIF P2_StoperZaklTesnenia.Banner.OUT.Stlaceny AND P2_UzivatelPrihlaseny THEN
				Paletka[i].PAR.ID_Operatora:= 'E2';//UsersVizu.CisloPrihlasenejKarty_Panel2;
				P2_Vizu.ZobrazHL12_ST3:= FALSE;
				P2_StoperZaklTesnenia.CMD.Banner_LED_OFF:= TRUE;
				CAM8.STAV.OldRunCounter:= CAM8.STAV.RunCounter;
				CAM8.STAV.Results_READY:= FALSE;
				SC_P2_StoperZaklTesnenia.ResetStep:= TRUE;
				SC_P2_StoperZaklTesnenia.Step:= 165;
			ELSIF P2_StoperZaklTesnenia.Banner.OUT.Stlaceny AND NOT P2_UzivatelPrihlaseny THEN
				Paletka[i].PAR.ID_Operatora:= '';
			END_IF

		165:
			SC_P2_StoperZaklTesnenia.StepName:='165 - Automaticky Rezim - kamerova kontrola QR kodu PowerCP CAM8';//CAM 8
			SC_P2_StoperZaklTesnenia.IdleTime.PT:= T#5s;
			SC_P2_StoperZaklTesnenia.AlarmTime.PT:= T#5s;

			P2_StoperZaklTesnenia.Banner.IN.ModraLED_ON:= TRUE;

			IF NOT SC_P2_StoperZaklTesnenia.Switch1 THEN
				CAM8.CMD.Triger:= TRUE;
				SC_P2_StoperZaklTesnenia.IdleTime.IN:= TRUE;
				SC_P2_StoperZaklTesnenia.Switch1:= TRUE;
			END_IF

			IF CAM8.STAV.Results_READY AND CAM8.STAV.OldRunCounter <> CAM8.STAV.RunCounter THEN
				PocetTrigrovKamery:= 0;
				CAM8.STAV.Results_READY:= FALSE;
				CAM8.STAV.OldRunCounter:= CAM8.STAV.RunCounter;
				P2_StoperZaklTesnenia.CMD.Banner_LED_OFF:= TRUE;
				SC_P2_StoperZaklTesnenia.ResetStep:= TRUE;
				SC_P2_StoperZaklTesnenia.Step:= 168;
			ELSIF SC_P2_StoperZaklTesnenia.IdleTime.Q AND PocetTrigrovKamery < 5 THEN
				PocetTrigrovKamery:= PocetTrigrovKamery + 1;
				CAM8.STAV.Results_READY:= FALSE;
				CAM8.STAV.OldRunCounter:= CAM8.STAV.RunCounter;
				CAM8.CMD.Triger:= FALSE;
				P2_StoperZaklTesnenia.CMD.Banner_LED_OFF:= TRUE;
				SC_P2_StoperZaklTesnenia.ResetStep:= TRUE;
				SC_P2_StoperZaklTesnenia.Step:= 166;
			ELSIF SC_P2_StoperZaklTesnenia.IdleTime.Q AND PocetTrigrovKamery >= 5 THEN
				P2_Alarmy[292]:= TRUE;
				P2_Pracovisko.STAV.Porucha_ST1:= TRUE;
			END_IF

		166:
			SC_P2_StoperZaklTesnenia.StepName:='166 - Automaticky Rezim - cakam na opatovny triger kamery CAM8';
			SC_P2_StoperZaklTesnenia.IdleTime.PT:= T#1s;
			SC_P2_StoperZaklTesnenia.AlarmTime.PT:= T#5s;
			SC_P2_StoperZaklTesnenia.IdleTime.IN:= TRUE;

			IF SC_P2_StoperZaklTesnenia.IdleTime.Q THEN
				SC_P2_StoperZaklTesnenia.ResetStep:= TRUE;
				SC_P2_StoperZaklTesnenia.Step:= 165;
			END_IF

		168:
			SC_P2_StoperZaklTesnenia.StepName:='168 - Automaticky Rezim - vysledok kamerovej kontroly QR kodu Power CP';
			SC_P2_StoperZaklTesnenia.IdleTime.PT:= T#200ms;
			SC_P2_StoperZaklTesnenia.AlarmTime.PT:= T#5s;
			SC_P2_StoperZaklTesnenia.IdleTime.IN:= TRUE;

			IF Linka.P2_Kamery_OFF THEN
				CAM8.CMD.Triger:= FALSE;
				CAM8.PAR.ResultFotky:= 'PASS';
				SC_P2_StoperZaklTesnenia.ResetStep:= TRUE;
				SC_P2_StoperZaklTesnenia.Step:= 170;
			ELSIF NOT CAM8.STAV.BUSY AND SC_P2_StoperZaklTesnenia.IdleTime.Q THEN
				CAM8.CMD.Triger:= FALSE;
				IF CAM8.RESULT.PowerCP.CitanieQRkodu_PowerCP_OK THEN
					SC_P2_StoperZaklTesnenia.IdleTime.IN:= TRUE;
					IF SC_P2_StoperZaklTesnenia.IdleTime.Q THEN
						IF CAM8.RESULT.PowerCP.PrecitanyQRkod_PowerCP = Paletka[i].PAR.QRkodPowerCP THEN
							CAM8.PAR.ResultFotky:= 'PASS';
							SC_P2_StoperZaklTesnenia.ResetStep:= TRUE;
							SC_P2_StoperZaklTesnenia.Step:= 170;
						ELSE
							CAM8.PAR.ResultFotky:= 'FAIL';
							SC_P2_StoperZaklTesnenia.ResetStep:= TRUE;
							SC_P2_StoperZaklTesnenia.Step:= 170;
						END_IF
					END_IF
				ELSE
					CAM8.PAR.ResultFotky:= 'FAIL';
					SC_P2_StoperZaklTesnenia.ResetStep:= TRUE;
					SC_P2_StoperZaklTesnenia.Step:= 170;
				END_IF
			END_IF

		170:
			SC_P2_StoperZaklTesnenia.StepName:='170 - Automaticky Rezim - rozhodnutie podla kamerovej kontroly QR kodu Power CP';
			SC_P2_StoperZaklTesnenia.IdleTime.PT:= T#200ms;
			SC_P2_StoperZaklTesnenia.AlarmTime.PT:= T#5s;

			IF CAM8.PAR.ResultFotky = 'PASS' THEN
				CAM17.STAV.OldRunCounter:= CAM17.STAV.RunCounter;
				CAM17.STAV.Results_READY:= FALSE;
				SC_P2_StoperZaklTesnenia.ResetStep:= TRUE;
				SC_P2_StoperZaklTesnenia.Step:= 180;
			ELSIF CAM8.PAR.ResultFotky = 'FAIL' THEN
				SC_P2_StoperZaklTesnenia.ResetStep:= TRUE;
				SC_P2_StoperZaklTesnenia.Step:= 173;
			END_IF

		173:
			SC_P2_StoperZaklTesnenia.StepName:='173 - Automaticky Rezim - zobrazenie hlasenia neprecitany alebo odlisny QR kod Power CP, cakanie na rozhodnutie obsluhy';
			SC_P2_StoperZaklTesnenia.IdleTime.PT:= T#200ms;
			SC_P2_StoperZaklTesnenia.AlarmTime.PT:= T#5s;

			P2_StoperZaklTesnenia.Banner.IN.CervenaLED_ON:= Blikac500ms;

			IF NOT SC_P2_StoperZaklTesnenia.Switch1 THEN
				P2_Vizu.ZobrazHL10_ST3:= TRUE;
				SC_P2_StoperZaklTesnenia.Switch1:= TRUE;
			END_IF

			IF P2_StoperZaklTesnenia.Banner.OUT.Stlaceny THEN
				CAM8.STAV.Results_READY:= FALSE;
				CAM8.STAV.OldRunCounter:= CAM8.STAV.RunCounter;
				P2_Vizu.ZobrazHL10_ST3:= FALSE;
				P2_StoperZaklTesnenia.CMD.Banner_LED_OFF:= TRUE; //Zhasnem banner//
				SC_P2_StoperZaklTesnenia.ResetStep:= TRUE;
				SC_P2_StoperZaklTesnenia.Step:= 165;
			END_IF

		180:
			SC_P2_StoperZaklTesnenia.StepName:='180 - Automaticky Rezim - kamerova kontrola paletky CAM17'; //CAM 17//
			SC_P2_StoperZaklTesnenia.IdleTime.PT:= T#5s;
			SC_P2_StoperZaklTesnenia.AlarmTime.PT:= T#5s;

			P2_StoperZaklTesnenia.Banner.IN.ModraLED_ON:= TRUE;

			IF NOT SC_P2_StoperZaklTesnenia.Switch1 AND CAM17.STAV.Command_READY THEN
				CAM17.CMD.Triger:= TRUE;
				SC_P2_StoperZaklTesnenia.IdleTime.IN:= TRUE;
				SC_P2_StoperZaklTesnenia.Switch1:= TRUE;
			END_IF

			IF CAM17.STAV.Results_READY AND CAM17.STAV.Command_AKCEPTOVANY AND CAM17.STAV.OldRunCounter <> CAM17.STAV.RunCounter THEN
				PocetTrigrovKamery:= 0;
				CAM17.STAV.Results_READY:= FALSE;
				CAM17.STAV.OldRunCounter:= CAM17.STAV.RunCounter;
				P2_StoperZaklTesnenia.CMD.Banner_LED_OFF:= TRUE;
				SC_P2_StoperZaklTesnenia.ResetStep:= TRUE;
				SC_P2_StoperZaklTesnenia.Step:= 183;
			ELSIF SC_P2_StoperZaklTesnenia.IdleTime.Q AND PocetTrigrovKamery < 5 THEN
				PocetTrigrovKamery:= PocetTrigrovKamery + 1;
				CAM17.STAV.Results_READY:= FALSE;
				CAM17.STAV.OldRunCounter:= CAM17.STAV.RunCounter;
				CAM17.CMD.Triger:= FALSE;
				P2_StoperZaklTesnenia.CMD.Banner_LED_OFF:= TRUE;
				SC_P2_StoperZaklTesnenia.ResetStep:= TRUE;
				SC_P2_StoperZaklTesnenia.Step:= 181;
			ELSIF SC_P2_StoperZaklTesnenia.IdleTime.Q AND PocetTrigrovKamery >= 5 THEN
				P2_Alarmy[293]:= TRUE;
				P2_Pracovisko.STAV.Porucha_ST1:= TRUE;
			END_IF

		181:
			SC_P2_StoperZaklTesnenia.StepName:='181 - Automaticky Rezim - cakam na opatovny triger kamery CAM17';
			SC_P2_StoperZaklTesnenia.IdleTime.PT:= T#1s;
			SC_P2_StoperZaklTesnenia.AlarmTime.PT:= T#5s;

			SC_P2_StoperZaklTesnenia.IdleTime.IN:= TRUE;

			IF SC_P2_StoperZaklTesnenia.IdleTime.Q THEN
				SC_P2_StoperZaklTesnenia.ResetStep:= TRUE;
				SC_P2_StoperZaklTesnenia.Step:= 180;
			END_IF

		183:
			SC_P2_StoperZaklTesnenia.StepName:='183 - Automaticky Rezim - vysledok kamerovej kontroly paletky';
			SC_P2_StoperZaklTesnenia.IdleTime.PT:= T#500ms;
			SC_P2_StoperZaklTesnenia.AlarmTime.PT:= T#5s;
			SC_P2_StoperZaklTesnenia.IdleTime.IN:= TRUE;

			IF Linka.P2_Kamery_OFF THEN
				CAM17.CMD.Triger:= FALSE;
				CAM17.PAR.ResultFotky:= 'PASS';
				SC_P2_StoperZaklTesnenia.ResetStep:= TRUE;
				SC_P2_StoperZaklTesnenia.Step:= 185;
			ELSIF NOT CAM17.STAV.BUSY THEN
				CAM17.CMD.Triger:= FALSE;
				IF Linka.PAR.ZvolenyModel = '4F' THEN
					IF CAM17.RESULT.Paletka.Pritomn_Busbary_4F AND
						CAM17.RESULT.Paletka.Pritomn_PowerCP_4F AND
						CAM17.RESULT.Paletka.Pritomn_TopCoveru_4F AND
						CAM17.RESULT.Paletka.Pritomn_LavyMVcase AND
						CAM17.RESULT.Paletka.Pritomn_PravyMVcase AND
						CAM17.RESULT.Paletka.PrazdnaPoziciaTopCoveru THEN
						CAM17.PAR.ResultFotky:= 'PASS';
						SC_P2_StoperZaklTesnenia.ResetStep:= TRUE;
						SC_P2_StoperZaklTesnenia.Step:= 185;
					ELSE
						CAM17.PAR.ResultFotky:= 'FAIL';
						SC_P2_StoperZaklTesnenia.ResetStep:= TRUE;
						SC_P2_StoperZaklTesnenia.Step:= 185;
					END_IF
				ELSIF Linka.PAR.ZvolenyModel = '5F' THEN
					IF CAM17.RESULT.Paletka.Pritomn_Busbary_5F AND
						CAM17.RESULT.Paletka.Pritomn_PowerCP_5F AND
						CAM17.RESULT.Paletka.Pritomn_TopCoveru_5F AND
						CAM17.RESULT.Paletka.Pritomn_LavyMVcase AND
						CAM17.RESULT.Paletka.Pritomn_PravyMVcase AND
						CAM17.RESULT.Paletka.PrazdnaPoziciaTopCoveru THEN
						CAM17.PAR.ResultFotky:= 'PASS';
						SC_P2_StoperZaklTesnenia.ResetStep:= TRUE;
						SC_P2_StoperZaklTesnenia.Step:= 185;
					ELSE
						CAM17.PAR.ResultFotky:= 'FAIL';
						SC_P2_StoperZaklTesnenia.ResetStep:= TRUE;
						SC_P2_StoperZaklTesnenia.Step:= 185;
					END_IF
				ELSIF Linka.PAR.ZvolenyModel = '5H' THEN
					IF P2_StoperZaklTesnenia.STAV.ObsluhaOznacilaPaletku_NG THEN
						CAM17.PAR.ResultFotky:= 'FAIL';
						SC_P2_StoperZaklTesnenia.ResetStep:= TRUE;
						SC_P2_StoperZaklTesnenia.Step:= 540;
					ELSIF CAM17.RESULT.Paletka.Pritomn_Busbary_5H AND
						CAM17.RESULT.Paletka.Pritomn_PowerCP_5H AND
						CAM17.RESULT.Paletka.Pritomn_TopCoveru_5H AND
						CAM17.RESULT.Paletka.Pritomn_LavyMVcase AND
						CAM17.RESULT.Paletka.Pritomn_PravyMVcase AND
						CAM17.RESULT.Paletka.PrazdnaPoziciaTopCoveru THEN
						CAM17.PAR.ResultFotky:= 'PASS';
						SC_P2_StoperZaklTesnenia.ResetStep:= TRUE;
						SC_P2_StoperZaklTesnenia.Step:= 185;
					ELSE
						CAM17.PAR.ResultFotky:= 'FAIL';
						SC_P2_StoperZaklTesnenia.ResetStep:= TRUE;
						SC_P2_StoperZaklTesnenia.Step:= 185;
					END_IF
				END_IF
			END_IF

		185:
			SC_P2_StoperZaklTesnenia.StepName:='178 - Automaticky Rezim - rozhodnutie podla kamerovej kontroly paletky';
			SC_P2_StoperZaklTesnenia.IdleTime.PT:= T#200ms;
			SC_P2_StoperZaklTesnenia.AlarmTime.PT:= T#5s;

			IF CAM17.PAR.ResultFotky = 'PASS' THEN
				Paletka[i].PAR.StavPowerCP:= 'PASS';
				SC_P2_StoperZaklTesnenia.ResetStep:= TRUE;
				SC_P2_StoperZaklTesnenia.Step:= 540;
			ELSIF CAM17.PAR.ResultFotky = 'FAIL' THEN
				SC_P2_StoperZaklTesnenia.ResetStep:= TRUE;
				SC_P2_StoperZaklTesnenia.Step:= 187;
			END_IF

		187:
			SC_P2_StoperZaklTesnenia.StepName:='187 - Automaticky Rezim - zobrazenie hlasenia zle ulozeny material na paletke, cakam na potvrdenie bannerom';
			SC_P2_StoperZaklTesnenia.IdleTime.PT:= T#200ms;
			SC_P2_StoperZaklTesnenia.AlarmTime.PT:= T#5s;

			P2_StoperZaklTesnenia.Banner.IN.CervenaLED_ON:= Blikac500ms;

			IF NOT SC_P2_StoperZaklTesnenia.Switch1 THEN
				IF Linka.PAR.ZvolenyModel = '4F' THEN
					P2_Vizu.ZobrazHL1_ST3:= TRUE;
				ELSIF Linka.PAR.ZvolenyModel = '5F' THEN
					P2_Vizu.ZobrazHL2_ST3:= TRUE;
				ELSIF Linka.PAR.ZvolenyModel = '5H' THEN
					P2_Vizu.ZobrazHL3_ST3:= TRUE;
				END_IF
				SC_P2_StoperZaklTesnenia.Switch1:= TRUE;
			END_IF

			IF P2_StoperZaklTesnenia.Banner.OUT.Stlaceny THEN
				CAM17.STAV.Results_READY:= FALSE;
				P2_Vizu.ZobrazHL1_ST3:= FALSE;
				P2_Vizu.ZobrazHL2_ST3:= FALSE;
				P2_Vizu.ZobrazHL3_ST3:= FALSE;
				P2_StoperZaklTesnenia.CMD.Banner_LED_OFF:= TRUE;
				SC_P2_StoperZaklTesnenia.ResetStep:= TRUE;
				SC_P2_StoperZaklTesnenia.Step:= 190;
			ELSIF P2_ZaklTesn_KAM_Result_Ignoruj THEN
				CAM17.STAV.Results_READY:= FALSE;
				P2_ZaklTesn_KAM_Result_Ignoruj:= FALSE;
				Paletka[i].PAR.StavPowerCP:= 'PASS';
				Paletka[i].STAV.StavPaletky:= 'OK';
				P2_Vizu.ZobrazHL1_ST3:= FALSE;
				P2_Vizu.ZobrazHL2_ST3:= FALSE;
				P2_Vizu.ZobrazHL3_ST3:= FALSE;
				P2_StoperZaklTesnenia.CMD.Banner_LED_OFF:= TRUE;
				SC_P2_StoperZaklTesnenia.ResetStep:= TRUE;
				SC_P2_StoperZaklTesnenia.Step:= 540;
			END_IF

		190:
			SC_P2_StoperZaklTesnenia.StepName:='190 - Automaticky Rezim - vymazanie fotky kamery CAM17';
			SC_P2_StoperZaklTesnenia.IdleTime.PT:= T#200ms;
			SC_P2_StoperZaklTesnenia.AlarmTime.PT:= T#5s;

			IF Linka.KOM_FTP_OFF THEN
				SC_P2_StoperZaklTesnenia.ResetStep:= TRUE;
				SC_P2_StoperZaklTesnenia.Step:= 165;
			ELSIF NOT SC_P2_StoperZaklTesnenia.Switch1 THEN
				FTP_CAM17.CMD.VymazFotku:= TRUE;
				SC_P2_StoperZaklTesnenia.Switch1:= TRUE;
			END_IF

			IF FTP_CAM17.STATUS.KomunikaciaUkoncena THEN
				FTP_CAM17.CMD.VymazFotku:= FALSE;
				CAM8.STAV.Results_READY:= FALSE;
				CAM8.STAV.OldRunCounter:= CAM8.STAV.RunCounter;
				CAM17.STAV.Results_READY:= FALSE;
				CAM17.STAV.OldRunCounter:= CAM17.STAV.RunCounter;
				SC_P2_StoperZaklTesnenia.ResetStep:= TRUE;
				SC_P2_StoperZaklTesnenia.Step:= 165;
			ELSIF FTP_CAM17.STATUS.KomunikaciaError THEN
				P2_Alarmy[228]:= TRUE;
				P2_Pracovisko.STAV.Porucha_ST1:= TRUE;
			END_IF

			//******************************************Odoslanie fotiek na server******************************************//

		540:
			SC_P2_StoperZaklTesnenia.StepName:='540 - Automaticky Rezim - odoslanie fotky CAM 1 a CAM 17 na server Panasonic'; //CAM1 a CAM 17
			SC_P2_StoperZaklTesnenia.IdleTime.PT:= T#200ms;
			SC_P2_StoperZaklTesnenia.AlarmTime.PT:= T#5s;

			P2_StoperZaklTesnenia.Banner.IN.ModraRotujucaLED_ON:= TRUE;

			IF Linka.KOM_FTP_OFF THEN
				P2_StoperZaklTesnenia.CMD.Banner_LED_OFF:= TRUE;
				SC_P2_StoperZaklTesnenia.ResetStep:= TRUE;
				SC_P2_StoperZaklTesnenia.Step:= 550;
			ELSIF NOT SC_P2_StoperZaklTesnenia.Switch1 THEN
				FTP_CAM1.INPUTS.QRkodPowerCP:= Paletka[i].PAR.QRkodPowerCP;
				CisloFotky:= CisloFotky + 1;
				FTP_CAM1.INPUTS.IndexFotky:= USINT_TO_STRING(CisloFotky);
				FTP_CAM1.INPUTS.Result:= CAM1.PAR.ResultFotky;
				Reports.Kamery.P2_CAM1_KontrolaTesnenia:= CAM1.PAR.ResultFotky;

				FTP_CAM17.INPUTS.QRkodPowerCP:= Paletka[i].PAR.QRkodPowerCP;
				CisloFotky:= CisloFotky + 1;
				FTP_CAM17.INPUTS.IndexFotky:= USINT_TO_STRING(CisloFotky);
				FTP_CAM17.INPUTS.Result:= CAM17.PAR.ResultFotky;
				Reports.Kamery.P2_CAM17_KontrolaPaletky:= CAM17.PAR.ResultFotky;

				FTP_CAM1.CMD.OdosliFotku:= TRUE;
				FTP_CAM17.CMD.OdosliFotku:= TRUE;
				P2_ZakladanieTesnenia_Taktime.IN.START_MeraniaStratovehoCasu:= TRUE;
				SC_P2_StoperZaklTesnenia.Switch1:= TRUE;
			END_IF

			IF FTP_CAM1.STATUS.KomunikaciaUkoncena AND FTP_CAM17.STATUS.KomunikaciaUkoncena THEN
				P2_StoperZaklTesnenia.CMD.Banner_LED_OFF:= TRUE;
				FTP_CAM1.CMD.OdosliFotku:= FALSE;
				FTP_CAM17.CMD.OdosliFotku:= FALSE;
				P2_ZakladanieTesnenia_Taktime.IN.START_MeraniaStratovehoCasu:= FALSE;
				Paletka[i].STAV.OdoslanieFotiek_DONE:= TRUE;
				SC_P2_StoperZaklTesnenia.ResetStep:= TRUE;
				SC_P2_StoperZaklTesnenia.Step:= 550;
			ELSIF FTP_CAM1.STATUS.KomunikaciaError THEN
				P2_Alarmy[225]:= TRUE;
				P2_Pracovisko.STAV.Porucha_ST1:= TRUE;
			ELSIF FTP_CAM17.STATUS.KomunikaciaError THEN
				P2_Alarmy[228]:= TRUE;
				P2_Pracovisko.STAV.Porucha_ST1:= TRUE;
			END_IF

			//*****************************Odoslanie dát na server************************************//

		550:
			SC_P2_StoperZaklTesnenia.StepName:='550 - Automaticky Rezim - odoslanie stavu paletky na server';
			SC_P2_StoperZaklTesnenia.IdleTime.PT:= T#200ms;
			SC_P2_StoperZaklTesnenia.AlarmTime.PT:= T#10s;

			P2_StoperZaklTesnenia.Banner.IN.ModraRotujucaLED_ON:= TRUE;

			IF Linka.KOM_Panatrace_OFF THEN
				P2_StoperZaklTesnenia.CMD.Banner_LED_OFF:= TRUE;
				SC_P2_StoperZaklTesnenia.ResetStep:= TRUE;
				SC_P2_StoperZaklTesnenia.Step:= 560;
			ELSIF NOT SC_P2_StoperZaklTesnenia.Switch1 AND TRCB_P2_ZakladacTesnenia_ST3.STATUS.KOM_READY THEN
				TRCB_P2_ZakladacTesnenia_ST3.CMD.OdosliStavPaletky_TYP2:= TRUE;
				(*P2_ZakladanieTesnenia_Taktime.IN.START_MeraniaStratovehoCasu:= TRUE;*)
				SC_P2_StoperZaklTesnenia.Switch1:= TRUE;
			END_IF

			IF TRCB_P2_ZakladacTesnenia_ST3.STATUS.KomunikaciaUkoncena THEN
				P2_StoperZaklTesnenia.CMD.Banner_LED_OFF:= TRUE;
				TRCB_P2_ZakladacTesnenia_ST3.CMD.OdosliStavPaletky_TYP2:= FALSE;
				P2_ZakladanieTesnenia_Taktime.IN.START_MeraniaStratovehoCasu:= FALSE;
				SC_P2_StoperZaklTesnenia.ResetStep:= TRUE;
				SC_P2_StoperZaklTesnenia.Step:= 552;
			ELSIF TRCB_P2_ZakladacTesnenia_ST3.STATUS.KomunikaciaError THEN
				TRCB_P2_ZakladacTesnenia_ST3.CMD.OdosliStavPaletky_TYP2:= FALSE;
				P2_ZakladanieTesnenia_Taktime.IN.START_MeraniaStratovehoCasu:= FALSE;
				SC_P2_StoperZaklTesnenia.ResetStep:= TRUE;
				SC_P2_StoperZaklTesnenia.Step:= 557;
			END_IF

		552:
			SC_P2_StoperZaklTesnenia.StepName:='552 - Automaticky Rezim - kontrola odpovede servera';
			SC_P2_StoperZaklTesnenia.IdleTime.PT:= T#200ms;
			SC_P2_StoperZaklTesnenia.AlarmTime.PT:= T#10s;

			IF NOT TRCB_P2_ZakladacTesnenia_ST3.STATUS.KomunikaciaUkoncena THEN
				IF TRCB_P2_ZakladacTesnenia_ST3.OUTPUTS.PovolenieCinnostiNaPaletke = 'OK' THEN
					Paletka[i].STAV.Komunikacia_DONE:= TRUE;
					SC_P2_StoperZaklTesnenia.ResetStep:= TRUE;
					SC_P2_StoperZaklTesnenia.Step:= 560;
				ELSIF TRCB_P2_ZakladacTesnenia_ST3.OUTPUTS.PovolenieCinnostiNaPaletke = 'NG' THEN
					Paletka[i].STAV.QRkodFiltraPriradeny:= FALSE;
					Paletka[i].STAV.StavPaletky:= 'NG';
					SC_P2_StoperZaklTesnenia.ResetStep:= TRUE;
					SC_P2_StoperZaklTesnenia.Step:= 560;
				END_IF
			END_IF

		555:
			SC_P2_StoperZaklTesnenia.StepName:='555 - Automaticky Rezim - vyziadanie stavu komunikacie zo serverom';
			SC_P2_StoperZaklTesnenia.IdleTime.PT:= T#200ms;
			SC_P2_StoperZaklTesnenia.AlarmTime.PT:= T#10s;

			P2_StoperZaklTesnenia.Banner.IN.ModraRotujucaLED_ON:= TRUE;

			IF NOT SC_P2_StoperZaklTesnenia.Switch1 AND TRCB_P2_ZakladacTesnenia_ST3.STATUS.KOM_READY THEN
				TRCB_P2_ZakladacTesnenia_ST3.CMD.VyziadajStavPanatrace_TYP4:= TRUE;
				SC_P2_StoperZaklTesnenia.Switch1:= TRUE;
			END_IF

			IF TRCB_P2_ZakladacTesnenia_ST3.STATUS.KomunikaciaUkoncena THEN
				P2_StoperZaklTesnenia.CMD.Banner_LED_OFF:= TRUE;
				TRCB_P2_ZakladacTesnenia_ST3.CMD.VyziadajStavPanatrace_TYP4:= FALSE;
				SC_P2_StoperZaklTesnenia.ResetStep:= TRUE;
				SC_P2_StoperZaklTesnenia.Step:= 556;
			ELSIF TRCB_P2_ZakladacTesnenia_ST3.STATUS.KomunikaciaError THEN
				P2_StoperZaklTesnenia.CMD.Banner_LED_OFF:= TRUE;
				SC_P2_StoperZaklTesnenia.ResetStep:= TRUE;
				SC_P2_StoperZaklTesnenia.Step:= 557;
			END_IF

		556:
			SC_P2_StoperZaklTesnenia.StepName:='556 - Automaticky Rezim - kontrola odpovede servera';
			SC_P2_StoperZaklTesnenia.IdleTime.PT:= T#200ms;
			SC_P2_StoperZaklTesnenia.AlarmTime.PT:= T#5s;

			IF NOT TRCB_P2_ZakladacTesnenia_ST3.STATUS.KomunikaciaUkoncena THEN
				IF TRCB_P2_ZakladacTesnenia_ST3.OUTPUTS.DruhCinnostiNaPaletke = '0;Generating' THEN
					SC_P2_StoperZaklTesnenia.ResetStep:= TRUE;
					SC_P2_StoperZaklTesnenia.Step:= 557;
				ELSIF TRCB_P2_ZakladacTesnenia_ST3.OUTPUTS.DruhCinnostiNaPaletke = '1;Request' THEN
					SC_P2_StoperZaklTesnenia.ResetStep:= TRUE;
					SC_P2_StoperZaklTesnenia.Step:= 557;
				ELSIF TRCB_P2_ZakladacTesnenia_ST3.OUTPUTS.DruhCinnostiNaPaletke = '2;Report' THEN
					SC_P2_StoperZaklTesnenia.ResetStep:= TRUE;
					SC_P2_StoperZaklTesnenia.Step:= 550;
				ELSIF TRCB_P2_ZakladacTesnenia_ST3.OUTPUTS.DruhCinnostiNaPaletke = '3;Wedding' THEN
					SC_P2_StoperZaklTesnenia.ResetStep:= TRUE;
					SC_P2_StoperZaklTesnenia.Step:= 557;
				ELSIF TRCB_P2_ZakladacTesnenia_ST3.OUTPUTS.DruhCinnostiNaPaletke = '4;Status' THEN
					SC_P2_StoperZaklTesnenia.ResetStep:= TRUE;
					SC_P2_StoperZaklTesnenia.Step:= 557;
				ELSIF TRCB_P2_ZakladacTesnenia_ST3.OUTPUTS.DruhCinnostiNaPaletke = '5;' THEN
					SC_P2_StoperZaklTesnenia.ResetStep:= TRUE;
					SC_P2_StoperZaklTesnenia.Step:= 557;
				ELSE
					SC_P2_StoperZaklTesnenia.ResetStep:= TRUE;
					SC_P2_StoperZaklTesnenia.Step:= 557;
				END_IF
			END_IF

		557:
			SC_P2_StoperZaklTesnenia.StepName:='557 - Automaticky Rezim - rozhodnutie obsluhy po chybe komunikacie s Panatrace';
			SC_P2_StoperZaklTesnenia.IdleTime.PT:= T#200ms;
			SC_P2_StoperZaklTesnenia.AlarmTime.PT:= T#5s;

			P2_Vizu.ZobrazHL15_ST3:= TRUE;
            P2_StoperZaklTesnenia.CMD.Banner_LED_OFF:= TRUE;

			IF TRCB_P2_ZaklTesn_OpatovnyDopyt THEN
				TRCB_P2_ZaklTesn_OpatovnyDopyt:= FALSE;
				P2_Vizu.ZobrazHL15_ST3:= FALSE;
				SC_P2_StoperZaklTesnenia.ResetStep:= TRUE;
				SC_P2_StoperZaklTesnenia.Step:= 555;
			ELSIF TRCB_P2_ZaklTesn_PaletkaNG THEN
				TRCB_P2_ZaklTesn_PaletkaNG:= FALSE;
				P2_Vizu.ZobrazHL15_ST3:= FALSE;
				Paletka[i].STAV.StavPaletky := 'NG';
				Paletka[i].STAV.QRkodFiltraPriradeny:= FALSE;
				SC_P2_StoperZaklTesnenia.ResetStep:= TRUE;
				SC_P2_StoperZaklTesnenia.Step:= 560;
			END_IF

//		558:
//			SC_P2_StoperZaklTesnenia.StepName:='558 - Automaticky Rezim - vymazanie fotky kamery CAM17 a CAM1';
//			SC_P2_StoperZaklTesnenia.IdleTime.PT:= T#200ms;
//			SC_P2_StoperZaklTesnenia.AlarmTime.PT:= T#5s;
//
//			P2_StoperZaklTesnenia.Banner.IN.ModraRotujucaLED_ON:= TRUE;
//
//			IF NOT SC_P2_StoperZaklTesnenia.Switch1 THEN
//				FTP_CAM17.CMD.VymazFotku:= TRUE;
//				FTP_CAM1.CMD.VymazFotku:= TRUE;
//				SC_P2_StoperZaklTesnenia.Switch1:= TRUE;
//			END_IF
//
//			IF FTP_CAM17.STATUS.KomunikaciaUkoncena AND FTP_CAM1.STATUS.KomunikaciaUkoncena THEN
//				P2_StoperZaklTesnenia.CMD.Banner_LED_OFF:= TRUE;
//				FTP_CAM17.CMD.VymazFotku:= FALSE;
//				IF P2_StoperZaklTesnenia.STAV.ObsluhaOznacilaPaletku_NG THEN
//					SC_P2_StoperZaklTesnenia.ResetStep:= TRUE;
//					SC_P2_StoperZaklTesnenia.Step:= 560;
//				ELSE
//					SC_P2_StoperZaklTesnenia.ResetStep:= TRUE;
//					SC_P2_StoperZaklTesnenia.Step:= 105;
//				END_IF
//			ELSIF FTP_CAM17.STATUS.KomunikaciaError THEN
//				P2_Alarmy[228]:= TRUE;
//				P2_Pracovisko.STAV.Porucha_ST1:= TRUE;
//			ELSIF FTP_CAM1.STATUS.KomunikaciaError THEN
//				P2_Alarmy[225]:= TRUE;
//				P2_Pracovisko.STAV.Porucha_ST1:= TRUE;
//			END_IF

			//*************************************************Vyvezenie paletky*********************************************************************//

		560:
			SC_P2_StoperZaklTesnenia.StepName:='560 - Automaticky Rezim - cakam na vyvezenie na stoper maticovacky';
			SC_P2_StoperZaklTesnenia.IdleTime.PT:= T#1s;
			SC_P2_StoperZaklTesnenia.AlarmTime.PT:= T#5s;

			IF Paletka[i].STAV.StavPaletky = 'NG' THEN
				SC_P2_StoperZaklTesnenia.IdleTime.IN:= TRUE;
				P2_StoperZaklTesnenia.Banner.IN.CervenaLED_ON:= Blikac500ms;
			ELSE
				P2_StoperZaklTesnenia.Banner.IN.ZelenaLED_ON:= Blikac500ms;
			END_IF

			IF P2_StoperZaklTesnenia.KoniecCyklu THEN
				SC_P2_StoperZaklTesnenia.ResetStep:= TRUE;
				SC_P2_StoperZaklTesnenia.Step:= 0;
			ELSIF NOT P2_StoperMaticovacky.RFID_hlava.PritomnostPaletky AND
				SC_P2_StoperMaticovacky.Step = 100 AND
				NOT P2_StoperZaklTesnenia.STAV.PrebiehaVyvezeniePaletky AND
				(Paletka[i].STAV.StavPaletky <> 'NG' OR SC_P2_StoperZaklTesnenia.IdleTime.Q) THEN
				P2_StoperZaklTesnenia.CMD.Banner_LED_OFF:= TRUE;
				P2_StoperZaklTesnenia.OUT.ZasunStoper:= TRUE;
				P2_StoperZaklTesnenia.STAV.PrebiehaVyvezeniePaletky:= TRUE;
				SC_P2_StoperZaklTesnenia.ResetStep:= TRUE;
				SC_P2_StoperZaklTesnenia.Step:= 561;
			END_IF

		561:
			SC_P2_StoperZaklTesnenia.StepName:='561 - Automaticky Rezim - ukoncenie vyvazania na stoper maticovacky';
			SC_P2_StoperZaklTesnenia.IdleTime.PT:= T#200ms;
			SC_P2_StoperZaklTesnenia.AlarmTime.PT:= T#10s;

			SC_P2_StoperZaklTesnenia.AlarmTime.IN:= P2_StoperZaklTesnenia.RFID_hlava.PritomnostPaletky;

			SC_P2_StoperZaklTesnenia.IdleTime.IN:= NOT P2_StoperZaklTesnenia.RFID_hlava.PritomnostPaletky;

			IF NOT P2_StoperZaklTesnenia.RFID_hlava.PritomnostPaletky THEN
				TestovaciKus:= FALSE;
				CisloFotky:= 0;
				P2_StoperZaklTesnenia.PAR.StaryQRkod_Filtra5H:= Paletka[i].PAR.QRkodFiltra_5H;
				Paletka[i].PAR.StavPowerCP:= '';
				Paletka[i].STAV.Komunikacia_DONE:= FALSE;
				Paletka[i].STAV.OdoslanieFotiek_DONE:= FALSE;
				Paletka[i].STAV.QRkodFiltraPriradeny:= FALSE;
				Reports.Kamery.P2_CAM1_KontrolaTesnenia:= '';
				Reports.Kamery.P2_CAM17_KontrolaPaletky:= '';
				P2_StoperZaklTesnenia.OUT.ZasunStoper:= FALSE;
				P2_StoperZaklTesnenia.STAV.ObsluhaOznacilaPaletku_NG:= FALSE;
				SC_P2_StoperZaklTesnenia.ResetStep:= TRUE;
				SC_P2_StoperZaklTesnenia.Step:= 100;
			ELSIF SC_P2_StoperZaklTesnenia.AlarmTime.Q THEN
				P2_Alarmy[286]:= TRUE;
				P2_Pracovisko.STAV.Porucha_ST1:= TRUE;
			END_IF

			//*******************************************************Manuálny režim*******************************************************************************//
		700:
			SC_P2_StoperZaklTesnenia.StepName:='700 - Manualny Rezim';
			SC_P2_StoperZaklTesnenia.IdleTime.PT:= T#8s;
			SC_P2_StoperZaklTesnenia.AlarmTime.PT:= T#5s;

	END_CASE

				END_PROGRAM

PROGRAM _EXIT
				(* Insert code here *)

				END_PROGRAM
```

#### Variables.var - Local variables
```iecst
VAR
	PrecitanyQRkodPowerCP : STRING[80];
	PrecitanyQRkodFiltra5H : STRING[80];
	PrecitaneCisloPaletky : STRING[3];
	ServerOdpoved_StavPowerCP : STRING[5];
	i : USINT;
	TestovaciKus : BOOL;
	CisloFotky : USINT;
	PocetDopytovNaServer : USINT := 0;
	CisloFotky1 : USINT := 0;
	OpatovnaKontrolaFiltra_5H : BOOL := 0;
	PocetTrigrovKamery : USINT := 0;
END_VAR
```

#### IOLinkKomunikacia.st
```iecst
ACTION IOLinkKomunikacia:

	//RFID snímač paletky//
	P2_StoperZaklTesnenia.RFID_hlava();

	//Ovládanie bannera//
	P2_StoperZaklTesnenia.Banner.IN.Blikac100ms:= Blikac500ms;
	P2_StoperZaklTesnenia.Banner();

END_ACTION
```

### Program Logical/Program/Pracovisko_2/P2_ZaklTesnenia (IEC)
